Universal Robots PolyScope program: ability.urp

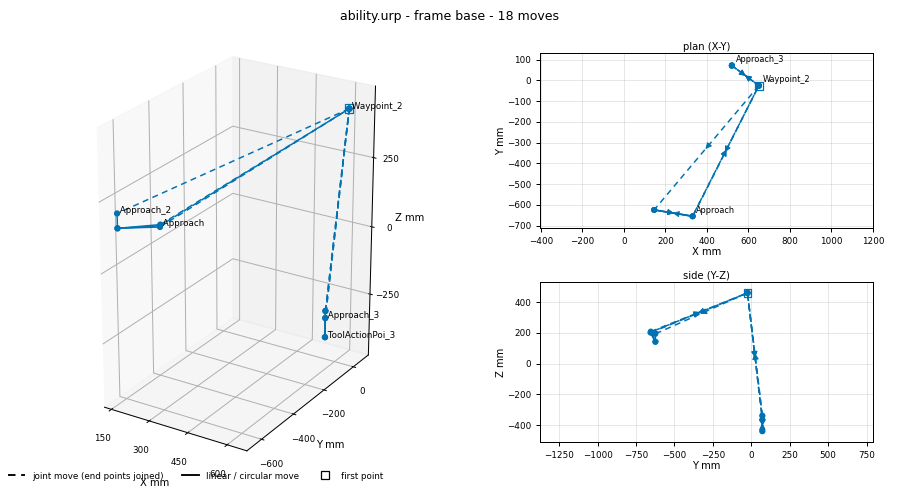
[picture p0: tool path of ability.urp in frame base, 18 of 18 moves have a stored position in this frame; points joined in program order, loops and branches not executed]
Program ability (installation=default directory=/programs createdIn=5.16.0 lastSavedIn=5.21.3 robotSerialNumber=20245590088)
Calibrated DH parameters: a=[0.000111, -0.242892, -0.343198, 0.000079, 0.000035, 0]; d=[0.162515, 160.798477, -193.665611, 33.000658, 0.099665, 0.099429]; alpha=[1.569849, -0.002171, 0.005777, 1.569501, -1.570045, 0]; deltaTheta=[0, -0.962932, 6.740777, 0.505346, 0, 0]
InitVariablesNode variables(variable(name=Pallet_2_cnt_1, expression=1), variable(name=Pallet_2_cnt_2, expression=1), variable(name=Pallet_2_cnt_3, expression=1), variable(name=Pallet_2_cnt_4, expression=1), variable(name=Pallet_2_lct_1, expression=1), variable(name=Pallet_2_lct_2, expression=1), variable(name=Pallet_2_lct_3, expression=1), variable(name=Pallet_2_lct_4, expression=1), variable(name=Pallet_2_lno_1, expression=1), variable(name=Pallet_2_lno_2, expression=1), variable(name=Pallet_2_lno_3, expression=1), variable(name=Pallet_2_lno_4, expression=1), variable(name=Pallet_2_sep_1, expression=False), variable(name=Pallet_2_sep_2, expression=False), variable(name=Pallet_2_sep_3, expression=False), variable(name=Pallet_2_sep_4, expression=False), variable(name=Pallet_2_tct_1, expression=1), variable(name=Pallet_2_tct_2, expression=1), variable(name=Pallet_2_tct_3, expression=1), variable(name=Pallet_2_tct_4, expression=1), variable(name=qNearApproach, expression=[0,0,0,0,0,0]), variable(name=qNearApproach_1, expression=[0,0,0,0,0,0]), variable(name=qNearApproach_2, expression=[0,0,0,0,0,0]), variable(name=qNearApproach_3, expression=[0,0,0,0,0,0]))
Robot Program (runOnlyOnce=false)
  SafeHome (positionOptionType=SPEED_AND_ACCELERATION speed=1.047198 acceleration=1.396263 nextMotionTime=2)
  URCap ER-Ability (EnabledRobotics - ER-ABILITY, Enabled Robotics ApS)
    'Insert event nodes here'
    URCap EventNode (EnabledRobotics - ER-ABILITY, Enabled Robotics ApS) dataModel(er_eventnode_inpname=calibrateFailed, er_eventnode_retvalname=none)
      Popup Message (haltProgram=false message=Calibrate to maker failed, marker not present inputType=Text)
    URCap EventNode (EnabledRobotics - ER-ABILITY, Enabled Robotics ApS) dataModel(er_eventnode_inpname=Gripper_Activate, er_eventnode_retvalname=none)
      URCap Gripper Activate (Robotiq_Grippers, Robotiq Inc.) dataModel(ResetAndActivateKey=false)
    URCap EventNode (EnabledRobotics - ER-ABILITY, Enabled Robotics ApS) dataModel(er_eventnode_inpname=Gripper_Open1, er_eventnode_retvalname=none)
      URCap Gripper (Robotiq_Grippers, Robotiq Inc.) dataModel(position=0.0, force=0.0, speed=100.0, positionInDouble=0.0, forceInDouble=0.0, speedInDouble=100.0, slaveIds=[9], blocking=true)
    URCap EventNode (EnabledRobotics - ER-ABILITY, Enabled Robotics ApS) dataModel(er_eventnode_inpname=Gripper_Close, er_eventnode_retvalname=none)
      URCap Gripper (Robotiq_Grippers, Robotiq Inc.) dataModel(position=100.0, force=0.0, speed=100.0, positionInDouble=100.0, forceInDouble=0.0, speedInDouble=100.0, slaveIds=[9], blocking=true)
    URCap EventNode (EnabledRobotics - ER-ABILITY, Enabled Robotics ApS) dataModel(er_eventnode_inpname=Unload, er_eventnode_retvalname=none, er_eventnode_input_arg_names=[arg_pose], er_eventnode_input_arg_types=[pose])
      Unload_ref := __er_Unload_arg_pose
      MoveJ speed 60 deg/s, acceleration 80 deg/s^2 (useActiveTCP=true optimoveEnabled=false optiMoveSpeed=0.3 optiMoveAcceleration=0.09) feature=Base
        Waypoint Waypoint_2: TCP in base x=650.372 y=-24.826 z=459.584 mm, rx=-2.156 ry=-0.0036 rz=-2.1951 rad; joints [154.293, -83.421, 119.183, -217.187, -61.732, 3.526] deg; TCP offset x=0 y=0 z=165 mm, rx=0 ry=0 rz=-1.57 rad
      URCap Palletizing (polyscope-pallet-impl, Universal Robots) dataModel(isPalletizing=true, palletFeature=Base, Length(key=objectHeight value=0.02 unit=M), Variable(key=qNearApproach, variable(name=qNearApproach, initializeExpression=[0,0,0,0,0,0])), Variable(key=name, variable(name=Pallet_2)), Variable(key=globalCountingVariable, variable(name=Pallet_2_cnt_1, initializeExpression=1)), Variable(key=layerCountingVariable, variable(name=Pallet_2_lct_1, initializeExpression=1)), Variable(key=layerNumberVariable, variable(name=Pallet_2_lno_1, initializeExpression=1)), Variable(key=handleSeparatorVariable, variable(name=Pallet_2_sep_1, initializeExpression=False)), Variable(key=totalCountVariable, variable(name=Pallet_2_tct_1, initializeExpression=1)), Variable(key=referencePoint, variable(featureName=referencePoint)), Variable(key=separatorPoint, variable(featureName=separatorPoint))); state(isChildrenLocked=true)
        URCap Patterns (polyscope-pallet-impl, Universal Robots) state(isChildrenLocked=true)
          URCap Pattern (polyscope-pallet-impl, Universal Robots) dataModel(UUID=a5dc391e-8dfa-4d41-8d42-d1a3ee492412, patternType=LINE, objects=3, Variable(key=nameVariable, variable(name=Line_Pattern_2))); state(isChildrenLocked=true)
            URCap Item (polyscope-pallet-impl, Universal Robots) dataModel(UUID=72ff3311-31d3-41c2-b996-3017bdb4fd84, patternType=LINE, index=0, calibrationDeltaTheta=[-2.9315277957084676E-8, -0.9629323736810536, 6.740777203655271, 0.5053459617643167, -4.967628234459065E-8, 1.3386501747369994E-8], calibrationA=[1.1102774445459327E-4, -0.24289161101812742, -0.3431982131897076, 7.864420289795527E-5, 3.464863415740183E-5, 0.0], calibrationD=[0.16251513683151333, 160.79847680046, -193.66561107659243, 33.000657595486956, 0.09966475034296075, 0.09942875700324125], calibrationAlpha=[1.5698494104941547, -0.002171092626713276, 0.005777151442641775, 1.5695009416808032, -1.570045005416207, 0.0], calibrationJointChecksum=[-1472934727, -1470672042, 693759659, -1457883488, -1458298026, -1457208209], calibrationStatus=2, calibrationValidChecksum=true, baseToFeature=[0.0, 0.0, 0.0, 0.0, 0.0, 0.0], TCPOffset=[2.775467002752441E-6, 1.4571326345524938E-7, 0.16500614774458194, 7.69911555341481E-6, 3.4900926535235165E-6, -1.5699764746901237], JointPositions(key=jointpositions, JointPosition(key=[1], Angle(key=pos value=3.019376 unit=RAD)), JointPosition(key=[2], Angle(key=pos value=-0.128164 unit=RAD)), JointPosition(key=[3], Angle(key=pos value=1.731691 unit=RAD)), JointPosition(key=[4], Angle(key=pos value=-3.173577 unit=RAD)), JointPosition(key=[5], Angle(key=pos value=-1.570163 unit=RAD)), JointPosition(key=[6], Angle(key=pos value=-0.124573 unit=RAD))), Variable(key=variable, variable(name=StartItem_2)))
            URCap Item (polyscope-pallet-impl, Universal Robots) dataModel(UUID=58fef9f4-1789-42d8-bc72-cd3fccb1f7d0, patternType=LINE, index=1, calibrationDeltaTheta=[-2.9315277957084676E-8, -0.9629323736810536, 6.740777203655271, 0.5053459617643167, -4.967628234459065E-8, 1.3386501747369994E-8], calibrationA=[1.1102774445459327E-4, -0.24289161101812742, -0.3431982131897076, 7.864420289795527E-5, 3.464863415740183E-5, 0.0], calibrationD=[0.16251513683151333, 160.79847680046, -193.66561107659243, 33.000657595486956, 0.09966475034296075, 0.09942875700324125], calibrationAlpha=[1.5698494104941547, -0.002171092626713276, 0.005777151442641775, 1.5695009416808032, -1.570045005416207, 0.0], calibrationJointChecksum=[-1472934727, -1470672042, 693759659, -1457883488, -1458298026, -1457208209], calibrationStatus=2, calibrationValidChecksum=true, baseToFeature=[0.0, 0.0, 0.0, 0.0, 0.0, 0.0], TCPOffset=[-3.781290865076392E-6, -1.8578380036826658E-5, 0.16498531422331186, 1.3351951116360783E-5, 2.5598841739530007E-5, -1.5700156061319748], JointPositions(key=jointpositions, JointPosition(key=[1], Angle(key=pos value=2.681982 unit=RAD)), JointPosition(key=[2], Angle(key=pos value=-0.129044 unit=RAD)), JointPosition(key=[3], Angle(key=pos value=1.711839 unit=RAD)), JointPosition(key=[4], Angle(key=pos value=-3.152808 unit=RAD)), JointPosition(key=[5], Angle(key=pos value=-1.570032 unit=RAD)), JointPosition(key=[6], Angle(key=pos value=-0.47729 unit=RAD))), Variable(key=variable, variable(name=EndItem_2)))
        URCap Layers (polyscope-pallet-impl, Universal Robots) dataModel(separators=[false], selectedPatterns=[a5dc391e-8dfa-4d41-8d42-d1a3ee492412])
        URCap At Each Item (polyscope-pallet-impl, Universal Robots) dataModel(selectedPattern=a5dc391e-8dfa-4d41-8d42-d1a3ee492412, selectedPosition=72ff3311-31d3-41c2-b996-3017bdb4fd84, Approach_calibrationDeltaTheta=[-2.9315277957084676E-8, -0.9629323736810536, 6.740777203655271, 0.5053459617643167, -4.967628234459065E-8, 1.3386501747369994E-8], Approach_calibrationA=[1.1102774445459327E-4, -0.24289161101812742, -0.3431982131897076, 7.864420289795527E-5, 3.464863415740183E-5, 0.0], Approach_calibrationD=[0.16251513683151333, 160.79847680046, -193.66561107659243, 33.000657595486956, 0.09966475034296075, 0.09942875700324125], Approach_calibrationAlpha=[1.5698494104941547, -0.002171092626713276, 0.005777151442641775, 1.5695009416808032, -1.570045005416207, 0.0], Approach_calibrationJointChecksum=[-1472934727, -1470672042, 693759659, -1457883488, -1458298026, -1457208209], Approach_calibrationStatus=2, Approach_calibrationValidChecksum=true, Approach_baseToFeature=[0.0, 0.0, 0.0, 0.0, 0.0, 0.0], Approach_TCPOffset=[-7.868968658605868E-6, 3.0566039674884138E-6, 0.1649950964573027, 8.399935251498573E-7, 1.7992186881394484E-5, -1.570036701188407], Exit_calibrationDeltaTheta=[-2.9315277957084676E-8, -0.9629323736810536, 6.740777203655271, 0.5053459617643167, -4.967628234459065E-8, 1.3386501747369994E-8], Exit_calibrationA=[1.1102774445459327E-4, -0.24289161101812742, -0.3431982131897076, 7.864420289795527E-5, 3.464863415740183E-5, 0.0], Exit_calibrationD=[0.16251513683151333, 160.79847680046, -193.66561107659243, 33.000657595486956, 0.09966475034296075, 0.09942875700324125], Exit_calibrationAlpha=[1.5698494104941547, -0.002171092626713276, 0.005777151442641775, 1.5695009416808032, -1.570045005416207, 0.0], Exit_calibrationJointChecksum=[-1472934727, -1470672042, 693759659, -1457883488, -1458298026, -1457208209], Exit_calibrationStatus=2, Exit_calibrationValidChecksum=true, Exit_baseToFeature=[0.0, 0.0, 0.0, 0.0, 0.0, 0.0], Exit_TCPOffset=[-1.1565336442947993E-5, 4.600903473428453E-6, 0.16499889588827082, 1.231938526291486E-5, -2.581973004009778E-5, -1.5700159038952088], currentWizardState=LANDING, Pose(key=refBaseToFeature, Position(key=posePosition, Length(key=X value=0 unit=M), Length(key=Y value=0 unit=M), Length(key=Z value=0 unit=M)), Rotation(key=poseRotation, Angle(key=RX value=0 unit=RAD), Angle(key=RY value=0 unit=RAD), Angle(key=RZ value=0 unit=RAD))), Pose(key=refPose, Position(key=posePosition, Length(key=X value=0.520227 unit=M), Length(key=Y value=0.071936 unit=M), Length(key=Z value=-0.439817 unit=M)), Rotation(key=poseRotation, Angle(key=RX value=3.14151 unit=RAD), Angle(key=RY value=0.015551 unit=RAD), Angle(key=RZ value=0.000011 unit=RAD))), JointPositions(key=Approach_jointpositions, JointPosition(key=[1], Angle(key=pos value=3.019748 unit=RAD)), JointPosition(key=[2], Angle(key=pos value=-0.306481 unit=RAD)), JointPosition(key=[3], Angle(key=pos value=1.868259 unit=RAD)), JointPosition(key=[4], Angle(key=pos value=-3.131259 unit=RAD)), JointPosition(key=[5], Angle(key=pos value=-1.569191 unit=RAD)), JointPosition(key=[6], Angle(key=pos value=-0.124391 unit=RAD))), JointPositions(key=Exit_jointpositions, JointPosition(key=[1], Angle(key=pos value=3.019838 unit=RAD)), JointPosition(key=[2], Angle(key=pos value=-0.373715 unit=RAD)), JointPosition(key=[3], Angle(key=pos value=1.911125 unit=RAD)), JointPosition(key=[4], Angle(key=pos value=-3.107472 unit=RAD)), JointPosition(key=[5], Angle(key=pos value=-1.569327 unit=RAD)), JointPosition(key=[6], Angle(key=pos value=-0.124086 unit=RAD))))
          URCap Generated Movements (polyscope-pallet-impl, Universal Robots) state(isChildrenLocked=true)
            MoveJ speed 60 deg/s, acceleration 80 deg/s^2 (useActiveTCP=true optimoveEnabled=false optiMoveSpeed=0.3 optiMoveAcceleration=0.09) feature=referencePoint
              Waypoint Approach_3: TCP in base x=520.075 y=72.086 z=-366.178 mm, rx=-3.1411 ry=-0.016 rz=0.0008 rad; joints [173.019, -17.56, 107.043, -179.408, -89.908, -7.127] deg; TCP offset x=-0.008 y=0.003 z=164.995 mm, rx=0 ry=0 rz=-1.57 rad; feature pose in base x=520.227 y=71.936 z=-439.817 mm, rx=3.1415 ry=0.0156 rz=0 rad
            MoveL speed 250 mm/s, acceleration 1200 mm/s^2 (useActiveTCP=true optimoveEnabled=false optiMoveSpeed=0.3 optiMoveAcceleration=0.09) feature(featureName=referencePoint)
              Waypoint ToolActionPoi_3: TCP in base x=520.227 y=71.936 z=-439.817 mm, rx=3.1415 ry=0.0156 rz=0 rad; joints [172.997, -7.343, 99.219, -181.833, -89.964, -7.137] deg; TCP offset x=0.003 y=0 z=165.006 mm, rx=0 ry=0 rz=-1.57 rad
            Folder Tool action
              URCap Gripper (Robotiq_Grippers, Robotiq Inc.) dataModel(position=100.0, force=100.0, speed=100.0, positionInDouble=100.0, forceInDouble=100.0, speedInDouble=100.0, slaveIds=[9], blocking=true)
            MoveL speed 250 mm/s, acceleration 1200 mm/s^2 (useActiveTCP=true optimoveEnabled=false optiMoveSpeed=0.3 optiMoveAcceleration=0.09) feature(featureName=referencePoint)
              Waypoint Exit_4: TCP in base x=520.222 y=71.948 z=-339.006 mm, rx=3.1415 ry=0.0156 rz=0 rad; joints [173.024, -21.412, 109.499, -178.045, -89.916, -7.11] deg; TCP offset x=-0.012 y=0.005 z=164.999 mm, rx=0 ry=0 rz=-1.57 rad
      MoveJ speed 60 deg/s, acceleration 80 deg/s^2 (useActiveTCP=true optimoveEnabled=false optiMoveSpeed=0.3 optiMoveAcceleration=0.09) feature=Base
        Waypoint Waypoint_2: TCP in base x=650.372 y=-24.826 z=459.584 mm, rx=-2.156 ry=-0.0036 rz=-2.1951 rad; joints [154.293, -83.421, 119.183, -217.187, -61.732, 3.526] deg; TCP offset x=0 y=0 z=165 mm, rx=0 ry=0 rz=-1.57 rad
      URCap Palletizing (polyscope-pallet-impl, Universal Robots) dataModel(isPalletizing=true, palletFeature=Unload_ref, Length(key=objectHeight value=0.02 unit=M), Variable(key=qNearApproach, variable(name=qNearApproach_1, initializeExpression=[0,0,0,0,0,0])), Variable(key=name, variable(name=Pallet_1)), Variable(key=globalCountingVariable, variable(name=Pallet_2_cnt_2, initializeExpression=1)), Variable(key=layerCountingVariable, variable(name=Pallet_2_lct_2, initializeExpression=1)), Variable(key=layerNumberVariable, variable(name=Pallet_2_lno_2, initializeExpression=1)), Variable(key=handleSeparatorVariable, variable(name=Pallet_2_sep_2, initializeExpression=False)), Variable(key=totalCountVariable, variable(name=Pallet_2_tct_2, initializeExpression=1)), Variable(key=referencePoint, variable(featureName=referencePoin_1)), Variable(key=separatorPoint, variable(featureName=separatorPoin_1))); state(isChildrenLocked=true)
        URCap Patterns (polyscope-pallet-impl, Universal Robots) state(isChildrenLocked=true)
          URCap Pattern (polyscope-pallet-impl, Universal Robots) dataModel(UUID=07243d7f-bf8f-4104-9bd3-73f99270b9f6, patternType=LINE, objects=3, Variable(key=nameVariable, variable(name=Line_Pattern_1))); state(isChildrenLocked=true)
            URCap Item (polyscope-pallet-impl, Universal Robots) dataModel(UUID=e6243a9f-c885-4ed6-8873-203569e74fdc, patternType=LINE, index=0, calibrationDeltaTheta=[-2.9315277957084676E-8, -0.9629323736810536, 6.740777203655271, 0.5053459617643167, -4.967628234459065E-8, 1.3386501747369994E-8], calibrationA=[1.1102774445459327E-4, -0.24289161101812742, -0.3431982131897076, 7.864420289795527E-5, 3.464863415740183E-5, 0.0], calibrationD=[0.16251513683151333, 160.79847680046, -193.66561107659243, 33.000657595486956, 0.09966475034296075, 0.09942875700324125], calibrationAlpha=[1.5698494104941547, -0.002171092626713276, 0.005777151442641775, 1.5695009416808032, -1.570045005416207, 0.0], calibrationJointChecksum=[-1472934727, -1470672042, 693759659, -1457883488, -1458298026, -1457208209], calibrationStatus=2, calibrationValidChecksum=true, baseToFeature=[0.23673981765789284, -0.611972183808765, 0.18903732227235456, -2.141026582984071, 2.2897807452097325, 0.016012414057338102], TCPOffset=[9.450929993104484E-6, 2.989998933555782E-6, 0.16499819525025852, -1.199062941364452E-5, -1.937393725705956E-6, -1.5699867065514344], JointPositions(key=jointpositions, JointPosition(key=[1], Angle(key=pos value=1.589886 unit=RAD)), JointPosition(key=[2], Angle(key=pos value=-1.175719 unit=RAD)), JointPosition(key=[3], Angle(key=pos value=1.56216 unit=RAD)), JointPosition(key=[4], Angle(key=pos value=-1.956496 unit=RAD)), JointPosition(key=[5], Angle(key=pos value=-1.56484 unit=RAD)), JointPosition(key=[6], Angle(key=pos value=0.072738 unit=RAD))), Variable(key=variable, variable(name=StartItem_1)))
            URCap Item (polyscope-pallet-impl, Universal Robots) dataModel(UUID=c4ba0ccc-1ea8-4b4a-a0e5-b351c685b141, patternType=LINE, index=1, calibrationDeltaTheta=[-2.9315277957084676E-8, -0.9629323736810536, 6.740777203655271, 0.5053459617643167, -4.967628234459065E-8, 1.3386501747369994E-8], calibrationA=[1.1102774445459327E-4, -0.24289161101812742, -0.3431982131897076, 7.864420289795527E-5, 3.464863415740183E-5, 0.0], calibrationD=[0.16251513683151333, 160.79847680046, -193.66561107659243, 33.000657595486956, 0.09966475034296075, 0.09942875700324125], calibrationAlpha=[1.5698494104941547, -0.002171092626713276, 0.005777151442641775, 1.5695009416808032, -1.570045005416207, 0.0], calibrationJointChecksum=[-1472934727, -1470672042, 693759659, -1457883488, -1458298026, -1457208209], calibrationStatus=2, calibrationValidChecksum=true, baseToFeature=[0.23673981765789284, -0.611972183808765, 0.18903732227235456, -2.141026582984071, 2.2897807452097325, 0.016012414057338102], TCPOffset=[7.669371193125794E-6, -3.297689358472411E-6, 0.16498784317780033, 1.98672481329163E-5, 1.36833597855774E-5, -1.569980005419673], JointPositions(key=jointpositions, JointPosition(key=[1], Angle(key=pos value=1.296694 unit=RAD)), JointPosition(key=[2], Angle(key=pos value=-1.225646 unit=RAD)), JointPosition(key=[3], Angle(key=pos value=1.637575 unit=RAD)), JointPosition(key=[4], Angle(key=pos value=-1.981979 unit=RAD)), JointPosition(key=[5], Angle(key=pos value=-1.564743 unit=RAD)), JointPosition(key=[6], Angle(key=pos value=-0.220355 unit=RAD))), Variable(key=variable, variable(name=EndItem_1)))
        URCap Layers (polyscope-pallet-impl, Universal Robots) dataModel(separators=[false], selectedPatterns=[07243d7f-bf8f-4104-9bd3-73f99270b9f6])
        URCap At Each Item (polyscope-pallet-impl, Universal Robots) dataModel(selectedPattern=07243d7f-bf8f-4104-9bd3-73f99270b9f6, selectedPosition=e6243a9f-c885-4ed6-8873-203569e74fdc, Approach_calibrationDeltaTheta=[-2.9315277957084676E-8, -0.9629323736810536, 6.740777203655271, 0.5053459617643167, -4.967628234459065E-8, 1.3386501747369994E-8], Approach_calibrationA=[1.1102774445459327E-4, -0.24289161101812742, -0.3431982131897076, 7.864420289795527E-5, 3.464863415740183E-5, 0.0], Approach_calibrationD=[0.16251513683151333, 160.79847680046, -193.66561107659243, 33.000657595486956, 0.09966475034296075, 0.09942875700324125], Approach_calibrationAlpha=[1.5698494104941547, -0.002171092626713276, 0.005777151442641775, 1.5695009416808032, -1.570045005416207, 0.0], Approach_calibrationJointChecksum=[-1472934727, -1470672042, 693759659, -1457883488, -1458298026, -1457208209], Approach_calibrationStatus=2, Approach_calibrationValidChecksum=true, Approach_baseToFeature=[0.41951857232416634, -0.6276001084527416, 0.19064087324443962, 2.298941266052505, -2.094963843603307, -0.026024890576082926], Approach_TCPOffset=[-1.0721172402361479E-6, 5.0607942906344405E-6, 0.1649848756045411, 1.9220935045796832E-5, 1.7733349406037467E-5, -1.569994096687021], Exit_calibrationDeltaTheta=[-2.9315277957084676E-8, -0.9629323736810536, 6.740777203655271, 0.5053459617643167, -4.967628234459065E-8, 1.3386501747369994E-8], Exit_calibrationA=[1.1102774445459327E-4, -0.24289161101812742, -0.3431982131897076, 7.864420289795527E-5, 3.464863415740183E-5, 0.0], Exit_calibrationD=[0.16251513683151333, 160.79847680046, -193.66561107659243, 33.000657595486956, 0.09966475034296075, 0.09942875700324125], Exit_calibrationAlpha=[1.5698494104941547, -0.002171092626713276, 0.005777151442641775, 1.5695009416808032, -1.570045005416207, 0.0], Exit_calibrationJointChecksum=[-1472934727, -1470672042, 693759659, -1457883488, -1458298026, -1457208209], Exit_calibrationStatus=2, Exit_calibrationValidChecksum=true, Exit_baseToFeature=[0.41951857232416634, -0.6276001084527416, 0.19064087324443962, 2.298941266052505, -2.094963843603307, -0.026024890576082926], Exit_TCPOffset=[2.512783842112398E-7, -6.292299156385184E-6, 0.164982798886549, 3.3963650715383825E-5, 7.3614499074614325E-6, -1.5700061521109205], currentWizardState=LANDING, Pose(key=refBaseToFeature, Position(key=posePosition, Length(key=X value=0.23674 unit=M), Length(key=Y value=-0.611972 unit=M), Length(key=Z value=0.189037 unit=M)), Rotation(key=poseRotation, Angle(key=RX value=-2.141027 unit=RAD), Angle(key=RY value=2.289781 unit=RAD), Angle(key=RZ value=0.016012 unit=RAD))), Pose(key=refPose, Position(key=posePosition, Length(key=X value=0.145742 unit=M), Length(key=Y value=-0.623712 unit=M), Length(key=Z value=0.141843 unit=M)), Rotation(key=poseRotation, Angle(key=RX value=-2.162913 unit=RAD), Angle(key=RY value=2.278464 unit=RAD), Angle(key=RZ value=0.000017 unit=RAD))), JointPositions(key=Approach_jointpositions, JointPosition(key=[1], Angle(key=pos value=1.854629 unit=RAD)), JointPosition(key=[2], Angle(key=pos value=-0.99282 unit=RAD)), JointPosition(key=[3], Angle(key=pos value=1.11845 unit=RAD)), JointPosition(key=[4], Angle(key=pos value=-1.69568 unit=RAD)), JointPosition(key=[5], Angle(key=pos value=-1.565563 unit=RAD)), JointPosition(key=[6], Angle(key=pos value=0.155136 unit=RAD))), JointPositions(key=Exit_jointpositions, JointPosition(key=[1], Angle(key=pos value=1.868555 unit=RAD)), JointPosition(key=[2], Angle(key=pos value=-0.99492 unit=RAD)), JointPosition(key=[3], Angle(key=pos value=1.134976 unit=RAD)), JointPosition(key=[4], Angle(key=pos value=-1.723755 unit=RAD)), JointPosition(key=[5], Angle(key=pos value=-1.600502 unit=RAD)), JointPosition(key=[6], Angle(key=pos value=0.189967 unit=RAD))))
          URCap Generated Movements (polyscope-pallet-impl, Universal Robots) state(isChildrenLocked=true)
            MoveJ speed 60 deg/s, acceleration 80 deg/s^2 (useActiveTCP=true optimoveEnabled=false optiMoveSpeed=0.3 optiMoveAcceleration=0.09) feature=referencePoin_1
              Waypoint Approach: TCP in base x=330.449 y=-654.703 z=204.316 mm, rx=2.3601 ry=-2.0736 rz=0 rad; joints [106.262, -56.884, 64.082, -97.155, -89.7, 8.889] deg; TCP offset x=-0.001 y=0.005 z=164.985 mm, rx=0 ry=0 rz=-1.57 rad; feature pose in base x=330.216 y=-654.763 z=146.676 mm, rx=2.3106 ry=-2.0735 rz=-0.0098 rad
            MoveL speed 250 mm/s, acceleration 1200 mm/s^2 (useActiveTCP=true optimoveEnabled=false optiMoveSpeed=0.3 optiMoveAcceleration=0.09) feature(featureName=referencePoin_1)
              Waypoint ToolActionPoint: TCP in base x=145.742 y=-623.712 z=141.843 mm, rx=-2.1628 ry=2.2784 rz=0 rad; joints [91.094, -67.364, 89.505, -112.099, -89.659, 4.168] deg; TCP offset x=0.009 y=0.003 z=164.998 mm, rx=0 ry=0 rz=-1.57 rad
            Folder Tool action
              URCap Gripper (Robotiq_Grippers, Robotiq Inc.) dataModel(position=0.0, force=100.0, speed=100.0, positionInDouble=0.0, forceInDouble=100.0, speedInDouble=100.0, slaveIds=[9], blocking=true)
            MoveL speed 250 mm/s, acceleration 1200 mm/s^2 (useActiveTCP=true optimoveEnabled=false optiMoveSpeed=0.3 optiMoveAcceleration=0.09) feature(featureName=referencePoin_1)
              Waypoint Exit_1: TCP in base x=331.325 y=-654.768 z=200.74 mm, rx=2.3106 ry=-2.0734 rz=-0.0097 rad; joints [107.06, -57.005, 65.029, -98.764, -91.702, 10.884] deg; TCP offset x=0 y=-0.006 z=164.983 mm, rx=0 ry=0 rz=-1.57 rad
      MoveJ speed 60 deg/s, acceleration 80 deg/s^2 (useActiveTCP=true optimoveEnabled=false optiMoveSpeed=0.3 optiMoveAcceleration=0.09) feature=Base
        Waypoint Waypoint_2: TCP in base x=650.372 y=-24.826 z=459.584 mm, rx=-2.156 ry=-0.0036 rz=-2.1951 rad; joints [154.293, -83.421, 119.183, -217.187, -61.732, 3.526] deg; TCP offset x=0 y=0 z=165 mm, rx=0 ry=0 rz=-1.57 rad
    URCap EventNode (EnabledRobotics - ER-ABILITY, Enabled Robotics ApS) dataModel(er_eventnode_inpname=Palletize, er_eventnode_retvalname=none, er_eventnode_input_arg_names=[arg_pose], er_eventnode_input_arg_types=[pose])
      Pallet_ref := __er_Palletize_arg_pose
      MoveJ speed 60 deg/s, acceleration 80 deg/s^2 (useActiveTCP=true optimoveEnabled=false optiMoveSpeed=0.3 optiMoveAcceleration=0.09) feature=Base
        SuppressedNode
          Waypoint Waypoint_6: TCP in base x=245.062 y=-588.705 z=186.234 mm, rx=0.1364 ry=-2.1189 rz=-2.2778 rad; joints [99.257, -67.966, 82.645, -100.78, -86.752, 4.555] deg; TCP offset x=0 y=0 z=165 mm, rx=-1.57 ry=0 rz=0 rad
        Waypoint Waypoint_2: TCP in base x=650.372 y=-24.826 z=459.584 mm, rx=-2.156 ry=-0.0036 rz=-2.1951 rad; joints [154.293, -83.421, 119.183, -217.187, -61.732, 3.526] deg; TCP offset x=0 y=0 z=165 mm, rx=0 ry=0 rz=-1.57 rad
      URCap Palletizing (polyscope-pallet-impl, Universal Robots) dataModel(isPalletizing=true, palletFeature=Pallet_ref, Length(key=objectHeight value=0.02 unit=M), Variable(key=qNearApproach, variable(name=qNearApproach_2, initializeExpression=[0,0,0,0,0,0])), Variable(key=name, variable(name=Pallet_3)), Variable(key=globalCountingVariable, variable(name=Pallet_2_cnt_3, initializeExpression=1)), Variable(key=layerCountingVariable, variable(name=Pallet_2_lct_3, initializeExpression=1)), Variable(key=layerNumberVariable, variable(name=Pallet_2_lno_3, initializeExpression=1)), Variable(key=handleSeparatorVariable, variable(name=Pallet_2_sep_3, initializeExpression=False)), Variable(key=totalCountVariable, variable(name=Pallet_2_tct_3, initializeExpression=1)), Variable(key=referencePoint, variable(featureName=referencePoin_6)), Variable(key=separatorPoint, variable(featureName=separatorPoin_6))); state(isChildrenLocked=true)
        URCap Patterns (polyscope-pallet-impl, Universal Robots) state(isChildrenLocked=true)
          URCap Pattern (polyscope-pallet-impl, Universal Robots) dataModel(UUID=07243d7f-bf8f-4104-9bd3-73f99270b9f6, patternType=LINE, objects=3, Variable(key=nameVariable, variable(name=Line_Pattern_5))); state(isChildrenLocked=true)
            URCap Item (polyscope-pallet-impl, Universal Robots) dataModel(UUID=e6243a9f-c885-4ed6-8873-203569e74fdc, patternType=LINE, index=0, calibrationDeltaTheta=[-2.9315277957084676E-8, -0.9629323736810536, 6.740777203655271, 0.5053459617643167, -4.967628234459065E-8, 1.3386501747369994E-8], calibrationA=[1.1102774445459327E-4, -0.24289161101812742, -0.3431982131897076, 7.864420289795527E-5, 3.464863415740183E-5, 0.0], calibrationD=[0.16251513683151333, 160.79847680046, -193.66561107659243, 33.000657595486956, 0.09966475034296075, 0.09942875700324125], calibrationAlpha=[1.5698494104941547, -0.002171092626713276, 0.005777151442641775, 1.5695009416808032, -1.570045005416207, 0.0], calibrationJointChecksum=[-1472934727, -1470672042, 693759659, -1457883488, -1458298026, -1457208209], calibrationStatus=2, calibrationValidChecksum=true, baseToFeature=[0.23673981765789284, -0.611972183808765, 0.18903732227235456, -2.141026582984071, 2.2897807452097325, 0.016012414057338102], TCPOffset=[9.450929993104484E-6, 2.989998933555782E-6, 0.16499819525025852, -1.199062941364452E-5, -1.937393725705956E-6, -1.5699867065514344], Variable(key=variable, variable(name=StartItem_5)), JointPositions(key=jointpositions, JointPosition(key=[1], Angle(key=pos value=1.589886 unit=RAD)), JointPosition(key=[2], Angle(key=pos value=-1.175719 unit=RAD)), JointPosition(key=[3], Angle(key=pos value=1.56216 unit=RAD)), JointPosition(key=[4], Angle(key=pos value=-1.956496 unit=RAD)), JointPosition(key=[5], Angle(key=pos value=-1.56484 unit=RAD)), JointPosition(key=[6], Angle(key=pos value=0.072738 unit=RAD))))
            URCap Item (polyscope-pallet-impl, Universal Robots) dataModel(UUID=c4ba0ccc-1ea8-4b4a-a0e5-b351c685b141, patternType=LINE, index=1, calibrationDeltaTheta=[-2.9315277957084676E-8, -0.9629323736810536, 6.740777203655271, 0.5053459617643167, -4.967628234459065E-8, 1.3386501747369994E-8], calibrationA=[1.1102774445459327E-4, -0.24289161101812742, -0.3431982131897076, 7.864420289795527E-5, 3.464863415740183E-5, 0.0], calibrationD=[0.16251513683151333, 160.79847680046, -193.66561107659243, 33.000657595486956, 0.09966475034296075, 0.09942875700324125], calibrationAlpha=[1.5698494104941547, -0.002171092626713276, 0.005777151442641775, 1.5695009416808032, -1.570045005416207, 0.0], calibrationJointChecksum=[-1472934727, -1470672042, 693759659, -1457883488, -1458298026, -1457208209], calibrationStatus=2, calibrationValidChecksum=true, baseToFeature=[0.23673981765789284, -0.611972183808765, 0.18903732227235456, -2.141026582984071, 2.2897807452097325, 0.016012414057338102], TCPOffset=[-2.3997290626276944E-6, -9.254975530281762E-6, 0.16499519045082972, 1.0556111519674915E-5, 2.9534904204817573E-6, -1.570002396573619], Variable(key=variable, variable(name=EndItem_5)), JointPositions(key=jointpositions, JointPosition(key=[1], Angle(key=pos value=1.296666 unit=RAD)), JointPosition(key=[2], Angle(key=pos value=-1.220363 unit=RAD)), JointPosition(key=[3], Angle(key=pos value=1.6455 unit=RAD)), JointPosition(key=[4], Angle(key=pos value=-1.995206 unit=RAD)), JointPosition(key=[5], Angle(key=pos value=-1.564737 unit=RAD)), JointPosition(key=[6], Angle(key=pos value=-0.22028 unit=RAD))))
        URCap Layers (polyscope-pallet-impl, Universal Robots) dataModel(separators=[false], selectedPatterns=[07243d7f-bf8f-4104-9bd3-73f99270b9f6])
        URCap At Each Item (polyscope-pallet-impl, Universal Robots) dataModel(selectedPattern=07243d7f-bf8f-4104-9bd3-73f99270b9f6, selectedPosition=e6243a9f-c885-4ed6-8873-203569e74fdc, Approach_calibrationDeltaTheta=[-2.9315277957084676E-8, -0.9629323736810536, 6.740777203655271, 0.5053459617643167, -4.967628234459065E-8, 1.3386501747369994E-8], Approach_calibrationA=[1.1102774445459327E-4, -0.24289161101812742, -0.3431982131897076, 7.864420289795527E-5, 3.464863415740183E-5, 0.0], Approach_calibrationD=[0.16251513683151333, 160.79847680046, -193.66561107659243, 33.000657595486956, 0.09966475034296075, 0.09942875700324125], Approach_calibrationAlpha=[1.5698494104941547, -0.002171092626713276, 0.005777151442641775, 1.5695009416808032, -1.570045005416207, 0.0], Approach_calibrationJointChecksum=[-1472934727, -1470672042, 693759659, -1457883488, -1458298026, -1457208209], Approach_calibrationStatus=2, Approach_calibrationValidChecksum=true, Approach_baseToFeature=[0.23673981765789284, -0.611972183808765, 0.18903732227235456, -2.141026582984071, 2.2897807452097325, 0.016012414057338102], Approach_TCPOffset=[9.495891565264314E-6, 8.369767002247563E-6, 0.16500465550890478, -7.325521899760681E-6, -6.086892211594123E-6, -1.569995281697695], Exit_calibrationDeltaTheta=[-2.9315277957084676E-8, -0.9629323736810536, 6.740777203655271, 0.5053459617643167, -4.967628234459065E-8, 1.3386501747369994E-8], Exit_calibrationA=[1.1102774445459327E-4, -0.24289161101812742, -0.3431982131897076, 7.864420289795527E-5, 3.464863415740183E-5, 0.0], Exit_calibrationD=[0.16251513683151333, 160.79847680046, -193.66561107659243, 33.000657595486956, 0.09966475034296075, 0.09942875700324125], Exit_calibrationAlpha=[1.5698494104941547, -0.002171092626713276, 0.005777151442641775, 1.5695009416808032, -1.570045005416207, 0.0], Exit_calibrationJointChecksum=[-1472934727, -1470672042, 693759659, -1457883488, -1458298026, -1457208209], Exit_calibrationStatus=2, Exit_calibrationValidChecksum=true, Exit_baseToFeature=[0.23673981765789284, -0.611972183808765, 0.18903732227235456, -2.141026582984071, 2.2897807452097325, 0.016012414057338102], Exit_TCPOffset=[5.925386180272163E-6, 4.091241161741088E-6, 0.16502720657378125, -4.031284870227352E-5, -3.582726072883789E-5, -1.569981020605123], currentWizardState=LANDING, Pose(key=refBaseToFeature, Position(key=posePosition, Length(key=X value=0.23674 unit=M), Length(key=Y value=-0.611972 unit=M), Length(key=Z value=0.189037 unit=M)), Rotation(key=poseRotation, Angle(key=RX value=-2.141027 unit=RAD), Angle(key=RY value=2.289781 unit=RAD), Angle(key=RZ value=0.016012 unit=RAD))), Pose(key=refPose, Position(key=posePosition, Length(key=X value=0.145742 unit=M), Length(key=Y value=-0.623712 unit=M), Length(key=Z value=0.141843 unit=M)), Rotation(key=poseRotation, Angle(key=RX value=-2.162913 unit=RAD), Angle(key=RY value=2.278464 unit=RAD), Angle(key=RZ value=0.000017 unit=RAD))), JointPositions(key=Approach_jointpositions, JointPosition(key=[1], Angle(key=pos value=1.58998 unit=RAD)), JointPosition(key=[2], Angle(key=pos value=-1.214816 unit=RAD)), JointPosition(key=[3], Angle(key=pos value=1.478378 unit=RAD)), JointPosition(key=[4], Angle(key=pos value=-1.833606 unit=RAD)), JointPosition(key=[5], Angle(key=pos value=-1.564902 unit=RAD)), JointPosition(key=[6], Angle(key=pos value=0.0721 unit=RAD))), JointPositions(key=Exit_jointpositions, JointPosition(key=[1], Angle(key=pos value=1.589999 unit=RAD)), JointPosition(key=[2], Angle(key=pos value=-1.22079 unit=RAD)), JointPosition(key=[3], Angle(key=pos value=1.460087 unit=RAD)), JointPosition(key=[4], Angle(key=pos value=-1.80934 unit=RAD)), JointPosition(key=[5], Angle(key=pos value=-1.564927 unit=RAD)), JointPosition(key=[6], Angle(key=pos value=0.071976 unit=RAD))))
          URCap Generated Movements (polyscope-pallet-impl, Universal Robots) state(isChildrenLocked=true)
            MoveJ speed 60 deg/s, acceleration 80 deg/s^2 (useActiveTCP=true optimoveEnabled=false optiMoveSpeed=0.3 optiMoveAcceleration=0.09) feature=referencePoin_6
              Waypoint Approach_2: TCP in base x=145.733 y=-623.703 z=193.586 mm, rx=-2.1629 ry=2.2785 rz=0 rad; joints [91.099, -69.604, 84.705, -105.058, -89.662, 4.131] deg; TCP offset x=0.009 y=0.008 z=165.005 mm, rx=0 ry=0 rz=-1.57 rad; feature pose in base x=145.742 y=-623.712 z=141.843 mm, rx=-2.1629 ry=2.2785 rz=0 rad
            MoveL speed 250 mm/s, acceleration 1200 mm/s^2 (useActiveTCP=true optimoveEnabled=false optiMoveSpeed=0.3 optiMoveAcceleration=0.09) feature(featureName=referencePoin_6)
              Waypoint ToolActionPoi_2: TCP in base x=145.742 y=-623.712 z=141.843 mm, rx=-2.1629 ry=2.2785 rz=0 rad; joints [91.094, -67.364, 89.505, -112.099, -89.659, 4.168] deg; TCP offset x=0.009 y=0.003 z=164.998 mm, rx=0 ry=0 rz=-1.57 rad
            Folder Tool action
              URCap Gripper (Robotiq_Grippers, Robotiq Inc.) dataModel(position=100.0, force=22.0, speed=60.0, positionInDouble=100.0, forceInDouble=22.0, speedInDouble=60.0, slaveIds=[9], blocking=true)
            MoveL speed 250 mm/s, acceleration 1200 mm/s^2 (useActiveTCP=true optimoveEnabled=false optiMoveSpeed=0.3 optiMoveAcceleration=0.09) feature(featureName=referencePoin_6)
              Waypoint Exit_3: TCP in base x=332.077 y=-653.506 z=208.569 mm, rx=2.3097 ry=-2.072 rz=-0.0096 rad; joints [107.176, -57.299, 64.358, -97.848, -91.782, 10.977] deg; TCP offset x=0 y=0 z=165 mm, rx=0 ry=0 rz=-1.57 rad; feature pose in base x=330.203 y=-655.036 z=146.797 mm, rx=2.3097 ry=-2.072 rz=-0.0096 rad
      MoveJ speed 60 deg/s, acceleration 80 deg/s^2 (useActiveTCP=true optimoveEnabled=false optiMoveSpeed=0.3 optiMoveAcceleration=0.09) feature=Base
        Waypoint Waypoint_2: TCP in base x=650.372 y=-24.826 z=459.584 mm, rx=-2.156 ry=-0.0036 rz=-2.1951 rad; joints [154.293, -83.421, 119.183, -217.187, -61.732, 3.526] deg
      URCap Palletizing (polyscope-pallet-impl, Universal Robots) dataModel(palletFeature=Base, isPalletizing=true, Length(key=objectHeight value=0.02 unit=M), Variable(key=qNearApproach, variable(name=qNearApproach_3, initializeExpression=[0,0,0,0,0,0])), Variable(key=name, variable(name=Pallet_4)), Variable(key=globalCountingVariable, variable(name=Pallet_2_cnt_4, initializeExpression=1)), Variable(key=layerCountingVariable, variable(name=Pallet_2_lct_4, initializeExpression=1)), Variable(key=layerNumberVariable, variable(name=Pallet_2_lno_4, initializeExpression=1)), Variable(key=handleSeparatorVariable, variable(name=Pallet_2_sep_4, initializeExpression=False)), Variable(key=totalCountVariable, variable(name=Pallet_2_tct_4, initializeExpression=1)), Variable(key=referencePoint, variable(featureName=referencePoin_7)), Variable(key=separatorPoint, variable(featureName=separatorPoin_7))); state(isChildrenLocked=true)
        URCap Patterns (polyscope-pallet-impl, Universal Robots) state(isChildrenLocked=true)
          URCap Pattern (polyscope-pallet-impl, Universal Robots) dataModel(UUID=a5dc391e-8dfa-4d41-8d42-d1a3ee492412, patternType=LINE, objects=3, Variable(key=nameVariable, variable(name=Line_Pattern_6))); state(isChildrenLocked=true)
            URCap Item (polyscope-pallet-impl, Universal Robots) dataModel(UUID=72ff3311-31d3-41c2-b996-3017bdb4fd84, patternType=LINE, index=0, calibrationDeltaTheta=[-2.9315277957084676E-8, -0.9629323736810536, 6.740777203655271, 0.5053459617643167, -4.967628234459065E-8, 1.3386501747369994E-8], calibrationA=[1.1102774445459327E-4, -0.24289161101812742, -0.3431982131897076, 7.864420289795527E-5, 3.464863415740183E-5, 0.0], calibrationD=[0.16251513683151333, 160.79847680046, -193.66561107659243, 33.000657595486956, 0.09966475034296075, 0.09942875700324125], calibrationAlpha=[1.5698494104941547, -0.002171092626713276, 0.005777151442641775, 1.5695009416808032, -1.570045005416207, 0.0], calibrationJointChecksum=[-1472934727, -1470672042, 693759659, -1457883488, -1458298026, -1457208209], calibrationStatus=2, calibrationValidChecksum=true, baseToFeature=[0.0, 0.0, 0.0, 0.0, 0.0, 0.0], TCPOffset=[2.775467002752441E-6, 1.4571326345524938E-7, 0.16500614774458194, 7.69911555341481E-6, 3.4900926535235165E-6, -1.5699764746901237], Variable(key=variable, variable(name=StartItem_6)), JointPositions(key=jointpositions, JointPosition(key=[1], Angle(key=pos value=3.019376 unit=RAD)), JointPosition(key=[2], Angle(key=pos value=-0.128164 unit=RAD)), JointPosition(key=[3], Angle(key=pos value=1.731691 unit=RAD)), JointPosition(key=[4], Angle(key=pos value=-3.173577 unit=RAD)), JointPosition(key=[5], Angle(key=pos value=-1.570163 unit=RAD)), JointPosition(key=[6], Angle(key=pos value=-0.124573 unit=RAD))))
            URCap Item (polyscope-pallet-impl, Universal Robots) dataModel(UUID=58fef9f4-1789-42d8-bc72-cd3fccb1f7d0, patternType=LINE, index=1, calibrationDeltaTheta=[-2.9315277957084676E-8, -0.9629323736810536, 6.740777203655271, 0.5053459617643167, -4.967628234459065E-8, 1.3386501747369994E-8], calibrationA=[1.1102774445459327E-4, -0.24289161101812742, -0.3431982131897076, 7.864420289795527E-5, 3.464863415740183E-5, 0.0], calibrationD=[0.16251513683151333, 160.79847680046, -193.66561107659243, 33.000657595486956, 0.09966475034296075, 0.09942875700324125], calibrationAlpha=[1.5698494104941547, -0.002171092626713276, 0.005777151442641775, 1.5695009416808032, -1.570045005416207, 0.0], calibrationJointChecksum=[-1472934727, -1470672042, 693759659, -1457883488, -1458298026, -1457208209], calibrationStatus=2, calibrationValidChecksum=true, baseToFeature=[0.0, 0.0, 0.0, 0.0, 0.0, 0.0], TCPOffset=[-3.781290865076392E-6, -1.8578380036826658E-5, 0.16498531422331186, 1.3351951116360783E-5, 2.5598841739530007E-5, -1.5700156061319748], Variable(key=variable, variable(name=EndItem_6)), JointPositions(key=jointpositions, JointPosition(key=[1], Angle(key=pos value=2.681982 unit=RAD)), JointPosition(key=[2], Angle(key=pos value=-0.129044 unit=RAD)), JointPosition(key=[3], Angle(key=pos value=1.711839 unit=RAD)), JointPosition(key=[4], Angle(key=pos value=-3.152808 unit=RAD)), JointPosition(key=[5], Angle(key=pos value=-1.570032 unit=RAD)), JointPosition(key=[6], Angle(key=pos value=-0.47729 unit=RAD))))
        URCap Layers (polyscope-pallet-impl, Universal Robots) dataModel(separators=[false], selectedPatterns=[a5dc391e-8dfa-4d41-8d42-d1a3ee492412])
        URCap At Each Item (polyscope-pallet-impl, Universal Robots) dataModel(selectedPattern=a5dc391e-8dfa-4d41-8d42-d1a3ee492412, selectedPosition=72ff3311-31d3-41c2-b996-3017bdb4fd84, Approach_calibrationDeltaTheta=[-2.9315277957084676E-8, -0.9629323736810536, 6.740777203655271, 0.5053459617643167, -4.967628234459065E-8, 1.3386501747369994E-8], Approach_calibrationA=[1.1102774445459327E-4, -0.24289161101812742, -0.3431982131897076, 7.864420289795527E-5, 3.464863415740183E-5, 0.0], Approach_calibrationD=[0.16251513683151333, 160.79847680046, -193.66561107659243, 33.000657595486956, 0.09966475034296075, 0.09942875700324125], Approach_calibrationAlpha=[1.5698494104941547, -0.002171092626713276, 0.005777151442641775, 1.5695009416808032, -1.570045005416207, 0.0], Approach_calibrationJointChecksum=[-1472934727, -1470672042, 693759659, -1457883488, -1458298026, -1457208209], Approach_calibrationStatus=2, Approach_calibrationValidChecksum=true, Approach_baseToFeature=[0.0, 0.0, 0.0, 0.0, 0.0, 0.0], Approach_TCPOffset=[-7.868968658605868E-6, 3.0566039674884138E-6, 0.1649950964573027, 8.399935251498573E-7, 1.7992186881394484E-5, -1.570036701188407], Exit_calibrationDeltaTheta=[-2.9315277957084676E-8, -0.9629323736810536, 6.740777203655271, 0.5053459617643167, -4.967628234459065E-8, 1.3386501747369994E-8], Exit_calibrationA=[1.1102774445459327E-4, -0.24289161101812742, -0.3431982131897076, 7.864420289795527E-5, 3.464863415740183E-5, 0.0], Exit_calibrationD=[0.16251513683151333, 160.79847680046, -193.66561107659243, 33.000657595486956, 0.09966475034296075, 0.09942875700324125], Exit_calibrationAlpha=[1.5698494104941547, -0.002171092626713276, 0.005777151442641775, 1.5695009416808032, -1.570045005416207, 0.0], Exit_calibrationJointChecksum=[-1472934727, -1470672042, 693759659, -1457883488, -1458298026, -1457208209], Exit_calibrationStatus=2, Exit_calibrationValidChecksum=true, Exit_baseToFeature=[0.0, 0.0, 0.0, 0.0, 0.0, 0.0], Exit_TCPOffset=[-1.1565336442947993E-5, 4.600903473428453E-6, 0.16499889588827082, 1.231938526291486E-5, -2.581973004009778E-5, -1.5700159038952088], currentWizardState=LANDING, Pose(key=refBaseToFeature, Position(key=posePosition, Length(key=X value=0 unit=M), Length(key=Y value=0 unit=M), Length(key=Z value=0 unit=M)), Rotation(key=poseRotation, Angle(key=RX value=0 unit=RAD), Angle(key=RY value=0 unit=RAD), Angle(key=RZ value=0 unit=RAD))), Pose(key=refPose, Position(key=posePosition, Length(key=X value=0.520227 unit=M), Length(key=Y value=0.071936 unit=M), Length(key=Z value=-0.439817 unit=M)), Rotation(key=poseRotation, Angle(key=RX value=3.14151 unit=RAD), Angle(key=RY value=0.015551 unit=RAD), Angle(key=RZ value=0.000011 unit=RAD))), JointPositions(key=Approach_jointpositions, JointPosition(key=[1], Angle(key=pos value=3.019748 unit=RAD)), JointPosition(key=[2], Angle(key=pos value=-0.306481 unit=RAD)), JointPosition(key=[3], Angle(key=pos value=1.868259 unit=RAD)), JointPosition(key=[4], Angle(key=pos value=-3.131259 unit=RAD)), JointPosition(key=[5], Angle(key=pos value=-1.569191 unit=RAD)), JointPosition(key=[6], Angle(key=pos value=-0.124391 unit=RAD))), JointPositions(key=Exit_jointpositions, JointPosition(key=[1], Angle(key=pos value=3.019838 unit=RAD)), JointPosition(key=[2], Angle(key=pos value=-0.373715 unit=RAD)), JointPosition(key=[3], Angle(key=pos value=1.911125 unit=RAD)), JointPosition(key=[4], Angle(key=pos value=-3.107472 unit=RAD)), JointPosition(key=[5], Angle(key=pos value=-1.569327 unit=RAD)), JointPosition(key=[6], Angle(key=pos value=-0.124086 unit=RAD))))
          URCap Generated Movements (polyscope-pallet-impl, Universal Robots) state(isChildrenLocked=true)
            MoveJ speed 60 deg/s, acceleration 80 deg/s^2 (useActiveTCP=true optimoveEnabled=false optiMoveSpeed=0.3 optiMoveAcceleration=0.09) feature=referencePoin_7
              Waypoint Approach_3: TCP in base x=520.075 y=72.086 z=-366.178 mm, rx=-3.1411 ry=-0.016 rz=0.0008 rad; joints [173.019, -17.56, 107.043, -179.408, -89.908, -7.127] deg; TCP offset x=-0.008 y=0.003 z=164.995 mm, rx=0 ry=0 rz=-1.57 rad; feature pose in base x=520.227 y=71.936 z=-439.817 mm, rx=3.1415 ry=0.0156 rz=0 rad
            MoveL speed 250 mm/s, acceleration 1200 mm/s^2 (useActiveTCP=true optimoveEnabled=false optiMoveSpeed=0.3 optiMoveAcceleration=0.09) feature(featureName=referencePoin_7)
              Waypoint ToolActionPoi_3: TCP in base x=520.227 y=71.936 z=-439.817 mm, rx=3.1415 ry=0.0156 rz=0 rad; joints [172.997, -7.343, 99.219, -181.833, -89.964, -7.137] deg; TCP offset x=0.003 y=0 z=165.006 mm, rx=0 ry=0 rz=-1.57 rad
            Folder Tool action
              URCap Gripper (Robotiq_Grippers, Robotiq Inc.) dataModel(position=0.0, force=22.0, speed=60.0, positionInDouble=0.0, forceInDouble=22.0, speedInDouble=60.0, slaveIds=[9], blocking=true)
            MoveL speed 250 mm/s, acceleration 1200 mm/s^2 (useActiveTCP=true optimoveEnabled=false optiMoveSpeed=0.3 optiMoveAcceleration=0.09) feature(featureName=referencePoin_7)
              Waypoint Exit_4: TCP in base x=520.222 y=71.948 z=-339.006 mm, rx=3.1415 ry=0.0156 rz=0 rad; joints [173.024, -21.412, 109.499, -178.045, -89.916, -7.11] deg; TCP offset x=-0.012 y=0.005 z=164.999 mm, rx=0 ry=0 rz=-1.57 rad
      MoveJ speed 60 deg/s, acceleration 80 deg/s^2 (useActiveTCP=true optimoveEnabled=false optiMoveSpeed=0.3 optiMoveAcceleration=0.09) feature=Base
        Waypoint Waypoint_2: TCP in base x=650.372 y=-24.826 z=459.584 mm, rx=-2.156 ry=-0.0036 rz=-2.1951 rad; joints [154.293, -83.421, 119.183, -217.187, -61.732, 3.526] deg; TCP offset x=0 y=0 z=165 mm, rx=0 ry=0 rz=-1.57 rad
